FUNCTION_BLOCK DigitalOutput
VAR_INPUT
	on					: BOOL;
END_VAR
VAR_OUTPUT
	output				: BOOL;
END_VAR

output 					:= on;

END_FUNCTION_BLOCK

(* stored: Version 1.1.0.1
   POU DigitalOutput: Id {2083ad13-3ca1-405f-88ac-d150cb014f89}, SpecialFunc None *)
